TYPE ES_SpesoreLastra_A_B :
STRUCT
	Lado_A_0Grados 						: LREAL ;
	Lado_B_180Grados 					: LREAL ;
END_STRUCT
END_TYPE

(* stored: Version 1.1.0.1, ProductVersion 3.1.4024.11
   DUT ES_SpesoreLastra_A_B: Id {1649206a-1251-4639-820d-00433c58eeae} *)
